(* IEC 61131-3 sources: com.logicals.lc3.webinar/RPMControl_Webinar/src_PRG_MQTT_Raspi4_ST, 3 files *)

(* ---- PRG_Raspi4_MQTTConnect.iecst ---- *)
/*
 * Raspi4
 * MQTTConnect Task
 */
PROGRAM PRG_Raspi4_MQTTConnect
   /*
    * PRG_Raspi4_MQTTConnect
    */
	VAR_EXTERNAL
    /*
     * Globaler TraceLevel
     */
     gui_TraceLevel : UINT;
	END_VAR
   /*
    * Status Verbindung zum Broker
    */
	VAR_EXTERNAL
		/*
		 * State und Channel vom Connect
		 */
		 MQTT_State   : MQTT_SUBSCRIBER_STATE;
		 MQTT_Channel : DINT;
	END_VAR

    VAR_EXTERNAL
        /*
         * Conecting Status an WebCon
         */
         gui_MQTTConnecting    : UINT; // Anzahl der Zyklen in MQTTConnecting
        /*
         * Conect und DisConnect Status an WebCon
         */
	     gui_MQTTConOkCycle    : UINT; // Anzahl der Zyklen bis MQTT Connect
	     gui_MQTTConNotOkCycle : UINT; // Anzahl der Zyklen wenn MQTT DisConnect
        /*
         * Conect Status an WebCon
         */
         gx_MQTTConOk      : BOOL;
    END_VAR

    VAR

    l_ConState : MQTT_SUBSCRIBER_STATE;

    l_RC       : MQTT_RC;
    ldi_Ch     : DINT;

    l_RC_Disconnect : MQTT_RC;

  END_VAR

   VAR
    /*
     * DiagnoseBits fuer RTS
     */
     lx_RTSInit     : BOOL;
     lx_RTSRun      : BOOL;
     lx_RTSShutDown : BOOL;
     lx_RTSTerm     : BOOL;
   END_VAR

   VAR
	 //
	 // Aus HCLib
     // Alle Verbindungen bedienen
     // Hier werden die Daten konkret verschickt!
     FB_Raspi4_MQTTConnect        : FB_MQTTConnect;
  END_VAR

  VAR
    /*
     * Der Datentyp enthaelt alle wesentlichen Informationen f�r die Basis-
     * Einstellungen von MQTT
     */
     l_MQTTInitKom    : DT_MQTT;
  END_VAR

 /*
  * Initialisierungsmerker
  */
  VAR
     FB_InitR_TRIG       : R_TRIG;
  END_VAR

  VAR
    /* Lokaler InitPuls im Baustein */
     lx_CycleInit : BOOL;

    /* Lokaler Puls im Baustein */
     lx_CyclePulse : BOOL;
    /* Lokaler Zyklustaktzaehler */
     li_CycleCount : INT;

    /* Lokaler InitZyklustaktzaehler */
     li_CycleCountInitVal : INT;
  END_VAR

  VAR
    lstr_PRGName      : STRING[30] := 'PRG_Raspi4_MQTTConnect';
    lui_TraceLevel    : UINT     := 5;

    lui_POU_UID       : UINT;                                      // Lokale POU-ID
    lstr_InstName     : STRING[30];
    lstr_POU_InstPath : STRING[128];                               // Lokale POU-ID
   END_VAR
 /*
  * -------------------------------------------------
  * Start SPS-Programm PRG_Raspi4_MQTTConnect
  * -------------------------------------------------
  */
 /*
  * InitZyklus setzen wenn MQTT aktiv gesetzt!
  */
  FB_InitR_TRIG(CLK := TRUE,Q => lx_CycleInit);

 /*
  * CyclePulse
  */
  lx_CyclePulse := NOT(lx_CyclePulse);

 /*
  * LifeTick bzw. ZyklusZaehler
  */
  li_CycleCount := li_CycleCount + 1;

   IF lx_CycleInit = TRUE THEN
       /*
        * Globalen TraceLevel uebernehmen
        */
       lui_TraceLevel := gui_TraceLevel;
      /*
       * PI-Name fuer GVL-Liste
       */
       lstr_InstName        := GET_CURRENT_PI_NAME();
       lstr_POU_InstPath    := lstr_PRGName;
       li_CycleCountInitVal := li_CycleCountInitVal + 1;
   END_IF;

    /*
     * Es wird ein MQTT_Connect aufgebaut
     * Wird fuer Publish/Subscribe verwendet!
     * NUR ein Connect je Resource zum Broker erlaubt!
     *
     * Im RTSTerm bzw. RTSShutdown MUSS der Connect Disconnected werden!
     */
     FB_Raspi4_MQTTConnect(vistr_InstPath                := lstr_InstName,
     	                    vistr_BrokerAddress          := l_MQTTInitKom.BrokerAdress,
                            vistr_ClientID               := l_MQTTInitKom.Raspi4ClientID,
                            vo_State                     => l_ConState,              // Status fuer Connect fuer alle zu oeffnenden Verbindungen (Pub/Sub) zum Broker
                            vo_RC                        => l_RC,                    // Status fuer Connect fuer alle zu oeffnenden Fehler (Pub/Sub) zum Broker
                            vodi_ch                      => ldi_Ch,                  // Status fuer Connect fuer alle zu oeffnenden Kanaele (Pub/Sub) zum Broker
                            voui_CycleCount_Connecting   => gui_MQTTConnecting,
                            voui_CycleCount_Connected    => gui_MQTTConOkCycle,      // Wert auch in WebCon
                            voui_CycleCount_NotConnected => gui_MQTTConNotOkCycle,   // Wert auch in WebCon
                            vox_MQTTConOk                => gx_MQTTConOk);           // Wert auch in WebCon
   /*
    * Ausgabe der Daten!
    */
    MQTT_State   := l_ConState;
    MQTT_Channel := ldi_ch;

   /*
    * Diagnosebits des RTS
    */
    RTSCycleInfo(Init     => lx_RTSInit,
  	             Run      => lx_RTSRun,
  	             Shutdown => lx_RTSShutDown,
  	             Term     => lx_RTSTerm);

   /*
    * Disconnect!
    * In RTS.CFG ShutDown Cycle von 3 Sekunden eintragen!
    */
    IF lx_RTSTerm = TRUE OR lx_RTSShutDown = TRUE THEN
     MQTT_Disconnect(ch := ldi_ch,
                     rc => l_RC_Disconnect);
     MQTT_State   := l_ConState;
     MQTT_Channel := -1;
    END_IF;

END_PROGRAM

(* ---- PRG_Raspi4_MQTTPublish_Header.iecst ---- *)
 /*
  * logi.cals GmbH
  * A-3100 St. Poelten
  * Europaplatz 7/1
  * Tel.: 0043-5-77147
  *
  * logi.cals automation solutions & services GmbH
  * D-40738 Langenfeld
  * Postfach 1306
  * Tel.: 0049-2173-91910
  *
  * Contact:
  * dieter.goltz@logicals.com
  *
  * History:
  * Created:
  * DG 2021-05-30 MQTT Header
  *
  * Modified:
  * DG 2021-05-30 MQTT Header
  */

 /*
  * Description
  * ===========
  */

 /*
  * Beschreibung
  * ============
  * MQTT Kommunikation
  * Publish Header
  *
  */

/*
 * Lokaler Test
 * ============
 * sudo mosquitto_sub -d -t test   - test = Name des Topic -> /GHaus       - Header
 *                                                            /GHaus/Value - Werte
 *
 * sudo mosquitto_pub -d -t test –m “Hello” - test = Name des Topic -> /GHaus       - Header
 *                                                                     /GHaus/Value - Werte
 *
 *                               -m "Hello" -> String der verschickt wird!
 */

/*
 * Publish des Header von Raspi4
 */
PROGRAM PRG_Raspi4_MQTTPublish_Header
    /*
	 * PRG_Raspi4_MQTTPublish_Header
	 */
    VAR_EXTERNAL
         MQTTHeader       : MQTTHeader;
    END_VAR

	VAR_EXTERNAL
		/*
		 * State und Channel vom Connect
		 */
		 MQTT_State   : MQTT_SUBSCRIBER_STATE;
		 MQTT_Channel : DINT;
	END_VAR

	VAR_EXTERNAL
    /*
     * Globaler TraceLevel
     */
     gui_TraceLevel : UINT;
	END_VAR

	VAR_EXTERNAL
    /*
     * Uhrzeit und Daten von TimeBaustein abholen
     * und auf Globale Var in Byte schreiben
     * Fuer MQTT
     */
  	 gb_RTSSeconds : BYTE;
 	 gb_RTSMinutes : BYTE;
	 gb_RTSHours   : BYTE;

	 gb_RTSDay         : BYTE;
	 gb_RTSMonth       : BYTE;
	 gb_RTSYearHByte   : BYTE;
	 gb_RTSYearLByte   : BYTE;

    END_VAR

   VAR
      FB_MQTT_PublishRaspi4      : FB_MQTT_Publish;
   END_VAR

  VAR
    /*
     * Der Datentyp enthaelt alle wesentlichen Initwerte f�r die MQTT-Kommunkation
     */
     l_MQTTInitKom         : DT_MQTT;
    /*
     * Status-Informationen
     */
     ldi_PublishLifeTick : DINT;
     lx_PublishOK        : BOOL;
     lui_IPVal1          : UINT;
     lui_IPVal2          : UINT;
     lui_IPVal3          : UINT;
     ldint_MQTTChannel   : DINT;
     ldint_MQTTCount     : DINT;
     ldint_MQTTrc        : DINT;
     lsint_MQTTState     : SINT;
     lx_MQTTENO          : BOOL;
     luint_MQTTLength    : UINT;
     lui_PubTick         : UINT;
  END_VAR

  VAR
    l_ConState : MQTT_SUBSCRIBER_STATE;
    ldi_ConCh  : DINT;
  END_VAR

  VAR
    lstr_PRGName   : STRING[30] := 'PRG_Raspi4_MQTTPublish_Header';
    lui_TraceLevel : UINT     := 5;
  END_VAR

  VAR
     FB_InitR_TRIG       : R_TRIG;
  END_VAR

  VAR
    /* Lokaler InitPuls im Baustein */
     lx_CycleInit : BOOL;

    /* Lokaler Puls im Baustein */
     lx_CyclePulse : BOOL;
    /* Lokaler Zyklustaktzaehler */
     li_CycleCount : INT;

    /* Lokaler InitZyklustaktzaehler */
     li_CycleCountInitVal : INT;
  END_VAR

 /*
  * InitZyklus setzen wenn MQTT aktiv gesetzt!
  */
  FB_InitR_TRIG(CLK := TRUE,Q => lx_CycleInit);
 /*
  * CyclePulse
  */
  lx_CyclePulse := NOT(lx_CyclePulse);

 /*
  * LifeTick bzw. ZyklusZaehler
  */
  li_CycleCount := li_CycleCount + 1;

  /*
   * Steuerung Publish / Subscribe ueber die Visu
   *
   * Publish
   * Welche Daten sollen an den Broker zurueckgeschickt werden
   * Subscribe
   * Welche Daten sollen geholt werden?
   */
   IF lx_CycleInit = TRUE THEN
      /*
       * Init Messages senden
       */
       lui_TraceLevel := gui_TraceLevel;
       li_CycleCountInitVal := li_CycleCountInitVal + 1;
   END_IF;
   /*
    * Daten von MQTTConnect
    */
    l_ConState := MQTT_State;
    ldi_ConCh  := MQTT_Channel;

    IF l_ConState = MQTT_SUBSCRIBER_STATE#CONNECTED THEN

   	   MQTTHeader.Second    := gb_RTSSeconds;
 	   MQTTHeader.Minute    := gb_RTSMinutes;
	   MQTTHeader.Hour      := gb_RTSHours;

	   MQTTHeader.Day       := gb_RTSDay;
	   MQTTHeader.Month     := gb_RTSMonth;
	   MQTTHeader.YearHByte := gb_RTSYearHByte;
	   MQTTHeader.YearLByte := gb_RTSYearLByte;

       MQTTHeader.IPVal3 := TO_BYTE(RIGHT(IN:= l_MQTTInitKom.Raspi4IPAdress, L := 1));
       MQTTHeader.IPVal2 := TO_BYTE(LEFT(RIGHT(IN:= l_MQTTInitKom.Raspi4IPAdress, L := 2),1));
       MQTTHeader.IPVal1 := TO_BYTE(LEFT(RIGHT(IN:= l_MQTTInitKom.Raspi4IPAdress, L := 3),1));

       FB_MQTT_PublishRaspi4(vi_MQTTHeader            := MQTTHeader,
                             vistr_IPAddr             := l_MQTTInitKom.Raspi4IPAdress,
                             vistr_BrokerIPAddr       := l_MQTTInitKom.BrokerAdress,
                             vix_Init                 := lx_CycleInit,
                             vi_State                 := l_ConState,
                             vdi_ch                   := ldi_ConCh,
       	                     vistr_BrokerPublishTopic := l_MQTTInitKom.Raspi4Topic,

                             vodi_PublishLifeTick    => ldi_PublishLifeTick,
                             vox_PublishOK           => lx_PublishOK,
                             voui_IPVal1             => lui_IPVal1,
                             voui_IPVal2             => lui_IPVal2,
                             voui_IPVal3             => lui_IPVal3,
                             vodint_MQTTChannel      => ldint_MQTTChannel,
                             vodint_MQTTCount        => ldint_MQTTCount,
                             vodint_MQTTrc           => ldint_MQTTrc,
                             vosint_MQTTState        => lsint_MQTTState,
                             vox_MQTTENO             => lx_MQTTENO,
                             vouint_MQTTLength       => luint_MQTTLength,
                             voui_PubTick            => lui_PubTick);
     END_IF;
END_PROGRAM

(* ---- PRG_Raspi4_MQTTPublish_IO.iecst ---- *)
   /*
  * logi.cals GmbH
  * A-3100 St. Poelten
  * Europaplatz 7/1
  * Tel.: 0043-5-77147
  *
  * logi.cals automation solutions & services GmbH
  * D-40738 Langenfeld
  * Postfach 1306
  * Tel.: 0049-2173-91910
  *
  * Contact:
  * dieter.goltz@logicals.com
  *
  * History:
  * Created:
  * DG 2021-05-30
  *
  * Modified:
  * DG 2021-05-30 IO
  */

 /*
  * Description
  * ===========
  */

 /*
  * Beschreibung
  * ============
  * MQTT Kommunikation
  * Publish Werte als Topics (IO)
  *
  * Austausch der aktuellen Daten mit dem Broker
  *
  */
 PROGRAM PRG_Raspi4_MQTTPublish_IO

   VAR_EXTERNAL
	    /* ProcessValue - Analogeingang_1 0..32767 unskaliert */
		gr_PV : REAL;
	    /* SetPoint     - Analogeingang_2 0..32767 unskaliert */
		gr_SP : REAL;
	    /* OutValue     - Analogausgang_1 0..32767 skaliert von 0..100% */
		gr_Y : REAL;
	    /* OutValue     - Ausgang Regler 0..100% wird skaliert auf 0..32767 */
		gr_PID_OUT : REAL;

	    /* ManualWert 0..100% */
		gr_Manual : REAL;

	    /* ProcessValue - Analogeingang_1 Skaliert 0..100%*/
		gr_PV_Scale : REAL;
	    /* SetPoint     - Analogeingang_2 Skaliert 0..100% */
		gr_SP_Scale : REAL;
	    /* OutValue     - Analogausgang_1 Skaliert 0..100% */
		gr_Y_Scale  : REAL;
        /*
         * Anzeige der Betriebsart 1Aus4
         */
        /* An Ausgang Ausgangswert = 0% */
        gx_ModeRPM0 : BOOL;
        /* An Ausgang Ausgangswert = 25% */
        gx_ModeRPM1 : BOOL;
        /* An Ausgang Ausgangswert = 50% */
        gx_ModeRPM2 : BOOL;
        /* An Ausgang SetPoint von Poti */
        gx_ModeRPM3 : BOOL;

        /* Blinkfunktion */
        gx_Flash : BOOL;
   END_VAR
  /*
   * PRG_Raspi4_MQTTPublish_IO
   */
   VAR_EXTERNAL
    /*
     * State und Channel vom Connect
     */
     MQTT_State   : MQTT_SUBSCRIBER_STATE;
     MQTT_Channel : DINT;
   END_VAR

   VAR_EXTERNAL
      /*
       * Globaler TraceLevel
       */
       gui_TraceLevel : UINT;
   END_VAR

  /*
   * Publish Topic / BOOL-Status von Topic
   */
   VAR
       FB_MQTT_Publish_IOBlink             : FB_MQTT_Publish_IO;

       FB_MQTT_Publish_IOValModeRPM0       : FB_MQTT_Publish_IO;
       FB_MQTT_Publish_IOValModeRPM1       : FB_MQTT_Publish_IO;
       FB_MQTT_Publish_IOValModeRPM2       : FB_MQTT_Publish_IO;
       FB_MQTT_Publish_IOValModeRPM3       : FB_MQTT_Publish_IO;

       FB_MQTT_Publish_IOValPV             : FB_MQTT_Publish_IOVal;
       FB_MQTT_Publish_IOValSP             : FB_MQTT_Publish_IOVal;
       FB_MQTT_Publish_IOValY              : FB_MQTT_Publish_IOVal;
       FB_MQTT_Publish_IOValManual         : FB_MQTT_Publish_IOVal;
       FB_MQTT_Publish_IOValPV_Scale       : FB_MQTT_Publish_IOVal;
       FB_MQTT_Publish_IOValSP_Scale       : FB_MQTT_Publish_IOVal;
       FB_MQTT_Publish_IOValY_Scale        : FB_MQTT_Publish_IOVal;

   END_VAR

  VAR
    /*
     * Der Datentyp enthaelt alle wesentlichen Informationen fuer die Basis-
     * Einstellungen von MQTT
     */
     l_MQTTInitKom    : DT_MQTT;
  END_VAR

  VAR
    l_ConState : MQTT_SUBSCRIBER_STATE;
    ldi_ConCh  : DINT;
  END_VAR

   VAR
    lstr_PRGName : STRING[30] := 'PRG_Raspi4_MQTTPublish_IO';
    lui_TraceLevel : UINT     := 5;
   END_VAR
 /*
  * Initialisierungsmerker
  */
  VAR
     FB_InitR_TRIG       : R_TRIG;
  END_VAR

  VAR
    /* Lokaler InitPuls im Baustein */
     lx_CycleInit        : BOOL;

    /* Lokaler Puls im Baustein */
     lx_CyclePulse       : BOOL;
    /* Lokaler Zyklustaktzaehler */
     li_CycleCount       : INT;

    /* Lokaler InitZyklustaktzaehler */
     li_CycleCountInitVal : INT;
  END_VAR

  /*
   * InitZyklus setzen wenn MQTT aktiv gesetzt!
   */
   FB_InitR_TRIG(CLK := TRUE,Q => lx_CycleInit);

   lui_TraceLevel := gui_TraceLevel;

  /*
   * CyclePulse
   */
   lx_CyclePulse := NOT(lx_CyclePulse);

  /*
   * LifeTick bzw. ZyklusZaehler
   */
   li_CycleCount := li_CycleCount + 1;
  /*
   * -------------------------------------------------
   * Start SPS-Programm PRG_Raspi4_MQTTPublish_IO
   * -------------------------------------------------
   */

  /*
   * Steuerung Publish_IO
   *
   * Publish
   * Welche Einzel-Daten sollen an den Broker geschickt werden
   */
   IF lx_CycleInit = TRUE THEN
       li_CycleCountInitVal := li_CycleCountInitVal + 1;
   END_IF;

   /*
    * Daten von MQTTConnect
    */
    l_ConState := MQTT_State;
    ldi_ConCh  := MQTT_Channel;

   /*
    * Kommt von MQTTConnect
    * Wert MUSS 6 sein!
    */
    IF l_ConState = MQTT_SUBSCRIBER_STATE#CONNECTED /* connected */ THEN

   /*
    * Blinkfunktion an gx_Out8
    */
    FB_MQTT_Publish_IOBlink(viui_TraceLevel            := lui_TraceLevel,
                            vix_PubIn                  := gx_Flash,
                            vistr_BrokerPublishTopicIO := l_MQTTInitKom.Raspi4TopicIOBlink,
                            vi_State                   := l_ConState,
                            vidi_Ch                    := ldi_ConCh);

   /*
    * Mode RPM 0
    */
    FB_MQTT_Publish_IOValModeRPM0(viui_TraceLevel            := lui_TraceLevel,
                                  vix_PubIn                  := gx_ModeRPM0,
                                  vistr_BrokerPublishTopicIO := l_MQTTInitKom.Raspi4TopicIOModeRPM0,
                                  vi_State                   := l_ConState,
                                  vidi_Ch                    := ldi_ConCh);

   /*
    * Mode RPM 1
    */
    FB_MQTT_Publish_IOValModeRPM1(viui_TraceLevel            := lui_TraceLevel,
                                  vix_PubIn                  := gx_ModeRPM1,
                                  vistr_BrokerPublishTopicIO := l_MQTTInitKom.Raspi4TopicIOModeRPM1,
                                  vi_State                   := l_ConState,
                                  vidi_Ch                    := ldi_ConCh);

   /*
    * Mode RPM 2
    */
    FB_MQTT_Publish_IOValModeRPM2(viui_TraceLevel            := lui_TraceLevel,
                                  vix_PubIn                  := gx_ModeRPM2,
                                  vistr_BrokerPublishTopicIO := l_MQTTInitKom.Raspi4TopicIOModeRPM2,
                                  vi_State                   := l_ConState,
                                  vidi_Ch                    := ldi_ConCh);

   /*
    * Mode RPM 3
    */
    FB_MQTT_Publish_IOValModeRPM3(viui_TraceLevel            := lui_TraceLevel,
                                  vix_PubIn                  := gx_ModeRPM3,
                                  vistr_BrokerPublishTopicIO := l_MQTTInitKom.Raspi4TopicIOModeRPM3,
                                  vi_State                   := l_ConState,
                                  vidi_Ch                    := ldi_ConCh);
   /*
    * PV
    */
    FB_MQTT_Publish_IOValPV(viui_TraceLevel            := lui_TraceLevel,
                            vir_PubIn                  := gr_PV,
                            vistr_BrokerPublishTopicIO := l_MQTTInitKom.Raspi4TopicIOPV,
                            vi_State                   := l_ConState,
                            vidi_Ch                    := ldi_ConCh);

   /*
    * SP
    */
    FB_MQTT_Publish_IOValSP(viui_TraceLevel            := lui_TraceLevel,
                            vir_PubIn                  := gr_SP,
                            vistr_BrokerPublishTopicIO := l_MQTTInitKom.Raspi4TopicIOSP,
                            vi_State                   := l_ConState,
                            vidi_Ch                    := ldi_ConCh);

   /*
    * Y
    */
    FB_MQTT_Publish_IOValY(viui_TraceLevel            := lui_TraceLevel,
                            vir_PubIn                  := gr_Y,
                            vistr_BrokerPublishTopicIO := l_MQTTInitKom.Raspi4TopicIOY,
                            vi_State                   := l_ConState,
                            vidi_Ch                    := ldi_ConCh);

   /*
    * PV_Scale
    */
    FB_MQTT_Publish_IOValPV_Scale(viui_TraceLevel            := lui_TraceLevel,
                                  vir_PubIn                  := gr_PV_Scale,
                                  vistr_BrokerPublishTopicIO := l_MQTTInitKom.Raspi4TopicIOPV_Scale,
                                  vi_State                   := l_ConState,
                                  vidi_Ch                    := ldi_ConCh);

   /*
    * SP_Scale
    */
    FB_MQTT_Publish_IOValSP_Scale(viui_TraceLevel            := lui_TraceLevel,
                                  vir_PubIn                  := gr_SP_Scale,
                                  vistr_BrokerPublishTopicIO := l_MQTTInitKom.Raspi4TopicIOSP_Scale,
                                  vi_State                   := l_ConState,
                                  vidi_Ch                    := ldi_ConCh);

   /*
    * Y = PID_OUT = Stellsignale des Reglers OHNE Skalierung 0..100%
    */
    FB_MQTT_Publish_IOValY_Scale(viui_TraceLevel            := lui_TraceLevel,
                                 vir_PubIn                  := gr_Y_Scale,
                                 vistr_BrokerPublishTopicIO := l_MQTTInitKom.Raspi4TopicIOY_Scale,
                                 vi_State                   := l_ConState,
                                 vidi_Ch                    := ldi_ConCh);
//
//   /*
//    * Manual
//    */
//    FB_MQTT_Publish_IOValManual(viui_TraceLevel            := lui_TraceLevel,
//                                 vir_PubIn                  := gr_Manual,
//                                 vistr_BrokerPublishTopicIO := l_MQTTInitKom.Raspi4TopicIOManual,
//                                 vi_State                   := l_ConState,
//                                 vidi_Ch                    := ldi_ConCh);
//
   END_IF;

  END_PROGRAM
